FUNCTION_BLOCK FB_DryingPhase

VAR_INPUT
	bExecute : BOOL;
END_VAR
VAR_OUTPUT
	bDryingDone : BOOL := FALSE;
	bDryingError : BOOL := FALSE;
END_VAR
VAR
	eDryState	: (IDLE, POSITION_M1, OPEN_AIR, WAITING_TIME, CLOSE_AIR, HOME_M1, DONE, ERROR); //Drying Phase internal States
	
	fbSolenoidControl : FB_SolenoidControl; //Solenoid control fb instance
	tonAirDryTime : ton; //Timer to run air trought stages
	
	bStart 	: BOOL := FALSE; //Start Flag	
	bMoveM1	: BOOL := FALSE; // M1 Vertical Motor Movement Flag
	bM1RightPosition	: BOOL := FALSE; // Make sure M1 is in the right position
	
	//HMI progress bar animation variables
	tStartTime : TIME := T#0S; // Drying start timestamp
	rElapsedTimeSec : REAL := 0.0; // Time passed in seconds
	rTotalEstimatedTimeSec : REAL := 0.0; // Total estimated time
	bProgressInitDone : BOOL := FALSE; // Estimation only once
	
END_VAR

IF NOT bStart THEN
	eDryState := IDLE;
	bStart := bExecute;
END_IF

//HMI Progress Bar Animation
IF bProgressInitDone AND (eDryState <> IDLE) AND (eDryState <> DONE) AND (eDryState <> ERROR) THEN
	rElapsedTimeSec := TO_REAL(TIME() - tStartTime) / 1000.0;
	GVL_HMI.HMIAnimation.rLoadBarDry := MIN(100.0, rElapsedTimeSec / rTotalEstimatedTimeSec * 100.0);
END_IF

CASE eDryState OF
	
	IDLE:
		// Reset Flags
		bDryingDone := FALSE; 
		bDryingError := FALSE;
		bMoveM1 := FALSE;
        IF bStart THEN
			//Start time calculation
			tStartTime := TIME();
			rTotalEstimatedTimeSec := EstimateTotalTime();
			bProgressInitDone := TRUE;
			// Provide HMI animation details
			GVL_HMI.HMIAnimation.eIconStateDry := E_IconState.InProgress;
			GVL_HMI.HMIAnimation.sLoadTextDry := 'Starting'; 
			GVL_HMI.HMIAnimation.rLoadBarDry  := 0;	
			// Move to next step
			eDryState := POSITION_M1;
        END_IF
	
	POSITION_M1:
		// Updating the HMI icon text
		GVL_HMI.HMIAnimation.sLoadTextDry  := 'Moving Motor';
		
		IF NOT bMoveM1 THEN // M1 Movement to dry position
			bMoveM1 := GVL_Motion.aMotors[1].MoveAbsolute(	rPosition := GVL_Settings.stMachineParam.aM1Position[2],
															rVelocity := GVL_Settings.stMachineParam.rM1Velocity,
															rAcc := GVL_Settings.stMachineParam.rM1Accleration,
															rDec := GVL_Settings.stMachineParam.rM1Deceleration
															);
		END_IF
		
		
		
		IF bMoveM1 THEN
			bMoveM1 := FALSE; // Reset Movement flag
			eDryState := OPEN_AIR; // Next step
		END_IF
	
	OPEN_AIR:
		bM1RightPosition := ABS(GVL_Motion.M1Motor.rActualPos - GVL_Settings.stMachineParam.aM1Position[2]) <= 2.0;
		// Check if the motor M1 is in the correct position
		IF bM1RightPosition THEN
			// Set air by solenoid position
			IF GVL_IO.gSetSolenoidControl.PressureUp() THEN
				eDryState := WAITING_TIME; // Move to next step
			END_IF
		ELSE
			bMoveM1 := FALSE; // Reset Movement flag
			eDryState := POSITION_M1;
		END_IF
	
	WAITING_TIME:
		// Updating the HMI icon text
		GVL_HMI.HMIAnimation.sLoadTextDry  := 'Drying';
		
		//fbSolenoidControl(bExecute := FALSE); //Resets solenoid position
		tonAirDryTime(in := TRUE, pt := GVL_Recipe.stActiveRecipe.stOtherParams.tAirDryTime); //Start timer
		IF tonAirDryTime.Q THEN
			eDryState := CLOSE_AIR;
		END_IF
		
	CLOSE_AIR:
		tonAirDryTime(in := FALSE); //Timer resets
		//fbSolenoidControl(bExecute := TRUE, eSolenoidSet := E_SolenoidSet.IDLE); //Set air by solenoid position
		IF GVL_IO.gSetSolenoidControl.Idle() THEN //IF fbSolenoidControl.bDone THEN
			bMoveM1 := FALSE;
			eDryState := HOME_M1; //moving to Done Step
		END_IF
		
	HOME_M1:
		// Updating the HMI icon text
		GVL_HMI.HMIAnimation.sLoadTextDry  := 'Homing Motor';
		
		IF NOT bMoveM1 THEN // M1 Movement to dry position
			bMoveM1 := GVL_Motion.aMotors[1].MoveAbsolute(	rPosition := GVL_Settings.stMachineParam.aM1Position[1],
															rVelocity := GVL_Settings.stMachineParam.rM1Velocity,
															rAcc := GVL_Settings.stMachineParam.rM1Accleration,
															rDec := GVL_Settings.stMachineParam.rM1Deceleration
															);
		END_IF
		
		
		
		IF bMoveM1 THEN
			bMoveM1 := FALSE; // Reset Movement flag
			eDryState := DONE; // Next step
		END_IF
		
		
	DONE:
		// Check if M1 was homed 
		bM1RightPosition := ABS(GVL_Motion.M1Motor.rActualPos - GVL_Settings.stMachineParam.aM1Position[1]) <= 2.0;
		IF bM1RightPosition THEN
			//HMI Icon animation
			GVL_HMI.HMIAnimation.eIconStateDry := E_IconState.Completed;
			GVL_HMI.HMIAnimation.sLoadTextDry  := 'Completed'; 
			GVL_HMI.HMIAnimation.rLoadBarDry   := 100;
			
			bDryingDone := TRUE; //Sucess flag
		ELSE
			bMoveM1 := FALSE; // Reset Movement flag
			eDryState := HOME_M1; // step back
		END_IF
		
			
	ERROR:
		//HMI Icon animation
		GVL_HMI.HMIAnimation.sLoadTextDry := 'Error'; 
		GVL_HMI.HMIAnimation.rLoadBarDry  := 0;
		GVL_HMI.HMIAnimation.eIconStateDry := E_IconState.Waiting;
		
		bDryingError := TRUE; //Error Flag

END_CASE

METHOD EstimateTotalTime : REAL
VAR
	rTotalTime : LREAL := 0.0;
    rDistance : LREAL;
    rVelocity : LREAL;
END_VAR
// --- Motor M1 movement (sequential) ---
rDistance := ABS(GVL_Settings.stMachineParam.aM1Position[2] - GVL_Settings.stMachineParam.aM1Position[3]); //From seal position up to dry position
rVelocity := GVL_Settings.stMachineParam.rM1Velocity;
IF rVelocity > 0 THEN
    rTotalTime := rTotalTime + rDistance / rVelocity;
END_IF

// --- Solenoid switching times (estimated 0.5s per switch) ---
rTotalTime := rTotalTime + 0.5 * 3; // open_air, close_air, reset

// --- Timer duration from recipe (AirDryTime) ---
rTotalTime := rTotalTime + TO_REAL(GVL_Recipe.stActiveRecipe.stOtherParams.tAirDryTime) / 1000.0;

EstimateTotalTime := rTotalTime;
END_METHOD

METHOD Reset : BOOL
VAR_INPUT
END_VAR
//output flags
bDryingDone  := FALSE;
bDryingError  := FALSE;

//state machine sequence
eDryState	:= IDLE;

//fb's and timers
//fbSolenoidControl(bExecute := FALSE);
tonAirDryTime(In := FALSE);

//initiation flags
bStart := FALSE; 
bMoveM1 := FALSE; 

//Progress bar variables
tStartTime := T#0S;
rElapsedTimeSec := 0.0;
rTotalEstimatedTimeSec := 0.0;
bProgressInitDone := FALSE;
GVL_HMI.HMIAnimation.rLoadBarDry := 0;

IF NOT bDryingDone AND NOT bDryingError THEN
	Reset := TRUE;
	RETURN;
ELSE
	Reset := FALSE;
END_IF
END_METHOD

END_FUNCTION_BLOCK

(* stored: Version 1.1.0.1, ProductVersion 3.1.4024.15
   POU FB_DryingPhase: Id {3fed5c2e-00c0-41f9-b86a-23cb950cee48}, SpecialFunc None
   Method EstimateTotalTime: Id {05ac8e4d-b1e3-4e8e-9944-a1369c6a61ae}
   Method Reset: Id {9c3cea04-676b-42b4-ac96-ce199a63ef22} *)
